(* IEC 61131-3 sources: Industry-PLC-LLM/data/PLCBEAD_repo/PLCBEAD_PLCEmbed-main/PLC-BEAD/Source/GEB/Network_IS_URLCHR, 1 file *)

(* ---- IS_URLCHR.ST ---- *)
FUNCTION IS_URLCHR:BOOL

	VAR_INPUT
		IN :	BYTE;
	END_VAR

	IS_URLCHR := ((IN>BYTE#47) AND (IN<BYTE#58)) OR ((IN>BYTE#64) AND (IN<BYTE#91)) OR ((IN>BYTE#96) AND (IN<BYTE#123)) OR (in=BYTE#126) OR (in=BYTE#95) OR (in=BYTE#45) OR (in=BYTE#46);

END_FUNCTION

PROGRAM program0
	VAR
		IN :	BYTE;
		CEIL5_OUT : BOOL;
	END_VAR

  	CEIL5_OUT := IS_URLCHR(IN);
END_PROGRAM
